(* IEC 61131-3 sources: astools/Data/ASTemplates/Default/Export Dialog/LogicalView/Libraries/FileIO, 3 files *)

(* ---- FileIO.typ ---- *)
TYPE
    fiDIR_READ_DATA		: STRUCT						(*directory read structure*)
        Filename		: ARRAY[0..259] OF USINT;		(*file name*)
        Date			: DATE_AND_TIME;				(*date and time*)
        Filelength		: UDINT;						(*file length*)
	END_STRUCT;

    fiDIR_READ_EX_DATA	: STRUCT						(*directory read extended structure*)
        Filename		: ARRAY[0..259] OF USINT;		(*file name*)
        Date			: DATE_AND_TIME;				(*date and time*)
        Filelength		: UDINT;						(*file length*)
        Mode			: UINT;							(*mode*)
	END_STRUCT;

	fiFILE_INFO			: STRUCT						(*file information structure*)
		size			: UDINT;						(*size of file [bytes]*)
		linkCnt			: UDINT;						(*link count*)
		accTime			: DATE_AND_TIME;				(*time of last access*)
		modTime			: DATE_AND_TIME;				(*time of last data modification*)
		chgTime			: DATE_AND_TIME;				(*time of last file status change*)
		reserved		: ARRAY[0..20] OF UDINT;		(*reserved for future use*)
	END_STRUCT;
END_TYPE

(* ---- FileIO.fun ---- *)
{REDUND_CONTEXT} {REDUND_UNREPLICABLE} FUNCTION_BLOCK FileCreate				(*creates a file; asynchronous execution*)
	VAR_INPUT
		enable		: BOOL;				(*enables execution*)
		pDevice		: UDINT;			(*device name given as a pointer*)
		pFile		: UDINT;			(*pointer to the file name*)
	END_VAR

	VAR
        i_state		: UINT;				(*internal variable*)
		i_result	: UINT;				(*internal variable*)
        i_tmp		: UDINT;			(*internal variable*)
	END_VAR

	VAR_OUTPUT
		status		: UINT;				(*execution status: ERR_OK, ERR_FUB_ENABLE_FALSE, ERR_FUB_BUSY, 0xXXXX = see help*)
		ident		: UDINT;			(*identifier of the created file*)
	END_VAR
END_FUNCTION_BLOCK

{REDUND_CONTEXT} {REDUND_UNREPLICABLE} FUNCTION_BLOCK FileOpen					(*opens a file; asynchronous execution*)
	VAR_INPUT
		enable		: BOOL;				(*enables execution*)
		pDevice		: UDINT;			(*device name given as a pointer*)
		pFile		: UDINT;			(*pointer to the file name*)
		mode		: USINT;			(*access mode (FILE_R, FILE_W, FILE_RW)*)
	END_VAR

	VAR
        i_state		: UINT;				(*internal variable*)
		i_result	: UINT;				(*internal variable*)
        i_tmp		: UDINT;			(*internal variable*)
	END_VAR

	VAR_OUTPUT
		status		: UINT;				(*execution status: ERR_OK, ERR_FUB_ENABLE_FALSE, ERR_FUB_BUSY, 0xXXXX = see help*)
		ident		: UDINT;			(*identifier of the created file*)
		filelen		: UDINT;			(*file length*)
	END_VAR
END_FUNCTION_BLOCK

{REDUND_CONTEXT} {REDUND_UNREPLICABLE} FUNCTION_BLOCK FileClose				(*closes an open file; asynchronous execution*)
	VAR_INPUT
		enable		: BOOL;				(*enables execution*)
		ident		: UDINT;			(*identifier of the created file*)
	END_VAR

	VAR
        i_state		: UINT;				(*internal variable*)
		i_result	: UINT;				(*internal variable*)
        i_tmp		: UDINT;			(*internal variable*)
	END_VAR

	VAR_OUTPUT
		status		: UINT;				(*execution status: ERR_OK, ERR_FUB_ENABLE_FALSE, ERR_FUB_BUSY, 0xXXXX = see help*)
	END_VAR
END_FUNCTION_BLOCK

{REDUND_CONTEXT} {REDUND_UNREPLICABLE} FUNCTION_BLOCK FileRead					(*reads from an open file; asynchronous execution*)
	VAR_INPUT
		enable		: BOOL;				(*enables execution*)
		ident		: UDINT;			(*identifier of the created file*)
		offset		: UDINT;			(*offset*)
		pDest		: UDINT;			(*pointer to the read buffer*)
		len			: UDINT;			(*length of bytes to read*)
	END_VAR

	VAR
        i_state		: UINT;				(*internal variable*)
		i_result	: UINT;				(*internal variable*)
        i_tmp		: UDINT;			(*internal variable*)
	END_VAR

	VAR_OUTPUT
		status		: UINT;				(*execution status: ERR_OK, ERR_FUB_ENABLE_FALSE, ERR_FUB_BUSY, 0xXXXX = see help*)
	END_VAR
END_FUNCTION_BLOCK

{REDUND_CONTEXT} {REDUND_UNREPLICABLE} FUNCTION_BLOCK FileReadEx				(*reads from an open file and returns the number of actually read bytes; asynchronous execution*)
	VAR_INPUT
		enable		: BOOL;				(*enables execution*)
		ident		: UDINT;			(*identifier of the created file*)
		offset		: UDINT;			(*offset*)
		pDest		: UDINT;			(*pointer to the read buffer*)
		len			: UDINT;			(*number of bytes to read*)
	END_VAR

	VAR
        i_state		: UINT;				(*internal variable*)
		i_result	: UINT;				(*internal variable*)
        i_tmp		: UDINT;			(*internal variable*)
	END_VAR

	VAR_OUTPUT
		status		: UINT;				(*execution status: ERR_OK, ERR_FUB_ENABLE_FALSE, ERR_FUB_BUSY, 0xXXXX = see help*)
		bytesread	: UDINT;			(*number of bytes read*)
	END_VAR
END_FUNCTION_BLOCK

{REDUND_CONTEXT} {REDUND_UNREPLICABLE} FUNCTION_BLOCK FileWrite				(*writes to a file; asynchronous execution*)
	VAR_INPUT
		enable		: BOOL;				(*enables execution*)
		ident		: UDINT;			(*identifier of the created file*)
		offset		: UDINT;			(*offset*)
		pSrc		: UDINT;			(*pointer to the write buffer*)
		len			: UDINT;			(*number of bytes to write*)
	END_VAR

	VAR
        i_state		: UINT;				(*internal variable*)
		i_result	: UINT;				(*internal variable*)
        i_tmp		: UDINT;			(*internal variable*)
	END_VAR

	VAR_OUTPUT
		status		: UINT;				(*execution status: ERR_OK, ERR_FUB_ENABLE_FALSE, ERR_FUB_BUSY, 0xXXXX = see help*)
	END_VAR
END_FUNCTION_BLOCK

{REDUND_CONTEXT} {REDUND_UNREPLICABLE} FUNCTION_BLOCK FileWriteEx				(*writes to a file; asynchronous execution*)
	VAR_INPUT
		enable		: BOOL;				(*enables execution*)
		ident		: UDINT;			(*identifier of the created file*)
		offset		: UDINT;			(*offset*)
		pSrc		: UDINT;			(*pointer to the write buffer*)
		len			: UDINT;			(*number of bytes to write*)
		option		: UDINT;			(*options*)
	END_VAR

	VAR
        i_state		: UINT;				(*internal variable*)
		i_result	: UINT;				(*internal variable*)
        i_tmp		: UDINT;			(*internal variable*)
	END_VAR

	VAR_OUTPUT
		status		: UINT;				(*execution status: ERR_OK, ERR_FUB_ENABLE_FALSE, ERR_FUB_BUSY, 0xXXXX = see help*)
	END_VAR
END_FUNCTION_BLOCK

{REDUND_CONTEXT} {REDUND_UNREPLICABLE} FUNCTION_BLOCK FileRename				(*renames files; asynchronous execution*)
	VAR_INPUT
		enable		: BOOL;				(*enables execution*)
		pDevice		: UDINT;			(*device name given as a pointer*)
		pName		: UDINT;			(*pointer to the file name*)
		pNewName	: UDINT;			(*pointer to the new file name*)
	END_VAR

	VAR
        i_state		: UINT;				(*internal variable*)
		i_result	: UINT;				(*internal variable*)
        i_tmp		: UDINT;			(*internal variable*)
	END_VAR

	VAR_OUTPUT
		status		: UINT;				(*execution status: ERR_OK, ERR_FUB_ENABLE_FALSE, ERR_FUB_BUSY, 0xXXXX = see help*)
	END_VAR
END_FUNCTION_BLOCK

{REDUND_CONTEXT} {REDUND_UNREPLICABLE} FUNCTION_BLOCK FileCopy					(*copies a file; asynchronous execution*)
	VAR_INPUT
		enable		: BOOL;				(*enables execution*)
		pSrcDev		: UDINT;			(*pointer to the source file device name*)
		pSrc		: UDINT;			(*pointer to the existing file name*)
		pDestDev	: UDINT;			(*pointer to the destination file device name*)
		pDest		: UDINT;			(*pointer to the copy file name*)
		option		: USINT;			(*copy option*)
	END_VAR

	VAR
        i_state		: UINT;				(*internal variable*)
		i_result	: UINT;				(*internal variable*)
        i_tmp		: UDINT;			(*internal variable*)
	END_VAR

	VAR_OUTPUT
		status		: UINT;				(*execution status: ERR_OK, ERR_FUB_ENABLE_FALSE, ERR_FUB_BUSY, 0xXXXX = see help*)
	END_VAR
END_FUNCTION_BLOCK

{REDUND_CONTEXT} {REDUND_UNREPLICABLE} FUNCTION_BLOCK FileDelete				(*deletes a file; asynchronous execution*)
	VAR_INPUT
		enable		: BOOL;				(*enables execution*)
		pDevice		: UDINT;			(*device name given as a pointer*)
		pName		: UDINT;			(*pointer to the file name*)
	END_VAR

	VAR
        i_state		: UINT;				(*internal variable*)
		i_result	: UINT;				(*internal variable*)
        i_tmp		: UDINT;			(*internal variable*)
	END_VAR

	VAR_OUTPUT
		status		: UINT;				(*execution status: ERR_OK, ERR_FUB_ENABLE_FALSE, ERR_FUB_BUSY, 0xXXXX = see help*)
	END_VAR
END_FUNCTION_BLOCK

{REDUND_CONTEXT} {REDUND_UNREPLICABLE} FUNCTION_BLOCK FileInfo					(*gets information about a file; asynchronous execution*)
	VAR_INPUT
		enable		: BOOL;				(*enables execution*)
		pDevice		: UDINT;			(*device name given as a pointer*)
		pName		: UDINT;			(*file name given as pointer*)
		pInfo		: UDINT;			(*file information (fiFILE_INFO) structure given as pointer*)
	END_VAR

	VAR
        i_state		: UINT;				(*internal variable*)
		i_result	: UINT;				(*internal variable*)
        i_tmp		: UDINT;			(*internal variable*)
	END_VAR

	VAR_OUTPUT
		status		: UINT;				(*execution status: ERR_OK, ERR_FUB_ENABLE_FALSE, ERR_FUB_BUSY, 0xXXXX = see help*)
	END_VAR
END_FUNCTION_BLOCK

{REDUND_CONTEXT} {REDUND_UNREPLICABLE} FUNCTION_BLOCK FileTruncate				(*truncates a file's length; asynchronous execution*)
	VAR_INPUT
		enable		: BOOL;				(*enables execution*)
		pDevice		: UDINT;			(*device name given as a pointer*)
		pName		: UDINT;			(*file name given as pointer*)
		newLength	: UDINT;			(*new length*)
	END_VAR

	VAR
        i_state		: UINT;				(*internal variable*)
		i_result	: UINT;				(*internal variable*)
        i_tmp		: UDINT;			(*internal variable*)
	END_VAR

	VAR_OUTPUT
		status		: UINT;				(*execution status: ERR_OK, ERR_FUB_ENABLE_FALSE, ERR_FUB_BUSY, 0xXXXX = see help*)
	END_VAR
END_FUNCTION_BLOCK

{REDUND_CONTEXT} {REDUND_UNREPLICABLE} FUNCTION_BLOCK DirCreate				(*creates a directory; asynchronous execution*)
	VAR_INPUT
		enable		: BOOL;				(*enables execution*)
		pDevice		: UDINT;			(*device name given as a pointer*)
		pName		: UDINT;			(*pointer to the directory name*)
	END_VAR

	VAR
        i_state		: UINT;				(*internal variable*)
		i_result	: UINT;				(*internal variable*)
        i_tmp		: UDINT;			(*internal variable*)
	END_VAR

	VAR_OUTPUT
		status		: UINT;				(*execution status: ERR_OK, ERR_FUB_ENABLE_FALSE, ERR_FUB_BUSY, 0xXXXX = see help*)
	END_VAR
END_FUNCTION_BLOCK

{REDUND_CONTEXT} {REDUND_UNREPLICABLE} FUNCTION_BLOCK DirOpen					(*opens a directory; asynchronous execution*)
	VAR_INPUT
		enable		: BOOL;				(*enables execution*)
		pDevice		: UDINT;			(*device name given as a pointer*)
		pName		: UDINT;			(*pointer to the directory name*)
	END_VAR

	VAR
        i_state		: UINT;				(*internal variable*)
		i_result	: UINT;				(*internal variable*)
        i_tmp		: UDINT;			(*internal variable*)
	END_VAR

	VAR_OUTPUT
		status		: UINT;				(*execution status: ERR_OK, ERR_FUB_ENABLE_FALSE, ERR_FUB_BUSY, 0xXXXX = see help*)
		ident		: UDINT;			(*identifier of the directory*)
	END_VAR
END_FUNCTION_BLOCK

{REDUND_CONTEXT} {REDUND_UNREPLICABLE} FUNCTION_BLOCK DirClose					(*closes a directory; asynchronous execution*)
	VAR_INPUT
		enable		: BOOL;				(*enables execution*)
		ident		: UDINT;			(*identifier of the directory*)
	END_VAR

	VAR
        i_state		: UINT;				(*internal variable*)
		i_result	: UINT;				(*internal variable*)
        i_tmp		: UDINT;			(*internal variable*)
	END_VAR

	VAR_OUTPUT
		status		: UINT;				(*execution status: ERR_OK, ERR_FUB_ENABLE_FALSE, ERR_FUB_BUSY, 0xXXXX = see help*)
	END_VAR
END_FUNCTION_BLOCK

{REDUND_CONTEXT} {REDUND_UNREPLICABLE} FUNCTION_BLOCK DirRead					(*reads the individual file names in a directory; asynchronous execution*)
	VAR_INPUT
		enable		: BOOL;				(*enables execution*)
		pDevice		: UDINT;			(*device name given as a pointer*)
		pPath		: UDINT;			(*pointer to the path string*)
		entry		: UDINT;			(*specifies which entry should be read*)
		option		: USINT;			(*specifies whether directory names or filenames should be read*)
		pData		: UDINT;			(*pointer to the memory area where the information is copied*)
		data_len	: UDINT;			(*length of the provided data area*)
	END_VAR

	VAR
        i_state		: UINT;				(*internal variable*)
		i_result	: UINT;				(*internal variable*)
        i_tmp		: UDINT;			(*internal variable*)
	END_VAR

	VAR_OUTPUT
		status		: UINT;				(*execution status: ERR_OK, ERR_FUB_ENABLE_FALSE, ERR_FUB_BUSY, 0xXXXX = see help*)
	END_VAR
END_FUNCTION_BLOCK

{REDUND_CONTEXT} {REDUND_UNREPLICABLE} FUNCTION_BLOCK DirReadEx				(*reads the individual file or directory names in a directory; asynchronous execution*)
	VAR_INPUT
		enable		: BOOL;				(*enables execution*)
		ident		: UDINT;			(*identifier of the directory*)
		pData		: UDINT;			(*pointer to the memory area where the information is copied*)
		data_len	: UDINT;			(*length of the available data area*)
	END_VAR

	VAR
        i_state		: UINT;				(*internal variable*)
		i_result	: UINT;				(*internal variable*)
        i_tmp		: UDINT;			(*internal variable*)
	END_VAR

	VAR_OUTPUT
		status		: UINT;				(*execution status: ERR_OK, ERR_FUB_ENABLE_FALSE, ERR_FUB_BUSY, 0xXXXX = see help*)
	END_VAR
END_FUNCTION_BLOCK

{REDUND_CONTEXT} {REDUND_UNREPLICABLE} FUNCTION_BLOCK DirInfo					(*gets information about a directory; asynchronous execution*)
	VAR_INPUT
		enable		: BOOL;				(*enables execution*)
		pDevice		: UDINT;			(*device name given as a pointer*)
		pPath		: UDINT;			(*pointer to the path (directory name)*)
	END_VAR

	VAR
        i_state		: UINT;				(*internal variable*)
		i_result	: UINT;				(*internal variable*)
        i_tmp		: UDINT;			(*internal variable*)
	END_VAR

	VAR_OUTPUT
		status		: UINT;				(*execution status: ERR_OK, ERR_FUB_ENABLE_FALSE, ERR_FUB_BUSY, 0xXXXX = see help*)
		dirnum		: UDINT;			(*number of subdirectories in this directory*)
		filenum		: UDINT;			(*number of files in this directory*)
	END_VAR
END_FUNCTION_BLOCK

{REDUND_CONTEXT} {REDUND_UNREPLICABLE} FUNCTION_BLOCK DirRename				(*renames directories; asynchronous execution*)
	VAR_INPUT
		enable		: BOOL;				(*enables execution*)
		pDevice		: UDINT;			(*device name given as a pointer*)
		pName		: UDINT;			(*pointer to the directory name*)
		pNewName	: UDINT;			(*pointer to the new directory name*)
	END_VAR

	VAR
        i_state		: UINT;				(*internal variable*)
		i_result	: UINT;				(*internal variable*)
        i_tmp		: UDINT;			(*internal variable*)
	END_VAR

	VAR_OUTPUT
		status		: UINT;				(*execution status: ERR_OK, ERR_FUB_ENABLE_FALSE, ERR_FUB_BUSY, 0xXXXX = see help*)
	END_VAR
END_FUNCTION_BLOCK

{REDUND_CONTEXT} {REDUND_UNREPLICABLE} FUNCTION_BLOCK DirCopy					(*copies a directory*)
	VAR_INPUT
		enable		: BOOL;				(*enables execution*)
		pSrcDev		: UDINT;			(*pointer to the source file device name*)
		pSrcDir		: UDINT;			(*pointer to the source directory name*)
		pDestDev	: UDINT;			(*pointer to the destination file device name*)
		pDestDir	: UDINT;			(*pointer to the destination directory name*)
		option		: USINT;			(*copy option*)
	END_VAR

	VAR
        i_state		: UINT;				(*internal variable*)
		i_result	: UINT;				(*internal variable*)
        i_tmp		: UDINT;			(*internal variable*)
	END_VAR

	VAR_OUTPUT
		status		: UINT;				(*execution status: ERR_OK, ERR_FUB_ENABLE_FALSE, 0xXXXX = see help*)
	END_VAR
END_FUNCTION_BLOCK

{REDUND_CONTEXT} {REDUND_UNREPLICABLE} FUNCTION_BLOCK DirDelete				(*deletes a directory; asynchronous execution*)
	VAR_INPUT
		enable		: BOOL;				(*enables execution*)
		pDevice		: UDINT;			(*device name given as a pointer*)
		pName		: UDINT;			(*pointer to the directory name*)
	END_VAR

	VAR
        i_state		: UINT;				(*internal variable*)
		i_result	: UINT;				(*internal variable*)
        i_tmp		: UDINT;			(*internal variable*)
	END_VAR

	VAR_OUTPUT
		status		: UINT;				(*execution status: ERR_OK, ERR_FUB_ENABLE_FALSE, ERR_FUB_BUSY, 0xXXXX = see help*)
	END_VAR
END_FUNCTION_BLOCK

{REDUND_CONTEXT} {REDUND_UNREPLICABLE} FUNCTION_BLOCK DirDeleteEx				(*deletes a directory (all files and subdirectories); asynchronous execution*)
	VAR_INPUT
		enable		: BOOL;				(*enables execution*)
		pDevice		: UDINT;			(*device name given as a pointer*)
		pName		: UDINT;			(*pointer to the directory name*)
	END_VAR

	VAR
        i_state		: UINT;				(*internal variable*)
		i_result	: UINT;				(*internal variable*)
        i_tmp		: UDINT;			(*internal variable*)
	END_VAR

	VAR_OUTPUT
		status		: UINT;				(*execution status: ERR_OK, ERR_FUB_ENABLE_FALSE, ERR_FUB_BUSY, 0xXXXX = see help*)
	END_VAR
END_FUNCTION_BLOCK

{REDUND_CONTEXT} {REDUND_UNREPLICABLE} FUNCTION_BLOCK SetAttributes			(*sets attributes; asynchronous execution*)
	VAR_INPUT
		enable		: BOOL;				(*enables execution*)
		pDevice		: UDINT;			(*device name given as a pointer*)
		pPath		: UDINT;			(*pointer to the path name (file or directory)*)
		attributes	: USINT;			(*attributes*)
		option		: USINT;			(*set options*)
	END_VAR

	VAR
        i_state		: UINT;				(*internal variable*)
		i_result	: UINT;				(*internal variable*)
        i_tmp		: UDINT;			(*internal variable*)
	END_VAR

	VAR_OUTPUT
		status		: UINT;				(*execution status: ERR_OK, ERR_FUB_ENABLE_FALSE, ERR_FUB_BUSY, 0xXXXX = see help*)
	END_VAR
END_FUNCTION_BLOCK

{REDUND_CONTEXT} {REDUND_UNREPLICABLE} FUNCTION_BLOCK GetAttributes			(*reads attributes; asynchronous execution*)
	VAR_INPUT
		enable		: BOOL;				(*enables execution*)
		pDevice		: UDINT;			(*device name given as a pointer*)
		pPath		: UDINT;			(*pointer to the path name (file or directory)*)
	END_VAR

	VAR
        i_state		: UINT;				(*internal variable*)
		i_result	: UINT;				(*internal variable*)
        i_tmp		: UDINT;			(*internal variable*)
	END_VAR

	VAR_OUTPUT
		status		: UINT;				(*execution status: ERR_OK, ERR_FUB_ENABLE_FALSE, ERR_FUB_BUSY, 0xXXXX = see help*)
		attributes	: USINT;			(*attributes*)
	END_VAR
END_FUNCTION_BLOCK

{REDUND_CONTEXT} {REDUND_UNREPLICABLE} FUNCTION_BLOCK DevMemInfo				(*determines a file device's memory information; asynchronous execution*)
	VAR_INPUT
		enable		: BOOL;				(*enables execution*)
		pDevice		: UDINT;			(*device name given as a pointer*)
	END_VAR

	VAR
        i_state		: UINT;				(*internal variable*)
		i_result	: UINT;				(*internal variable*)
        i_tmp		: UDINT;			(*internal variable*)
	END_VAR

	VAR_OUTPUT
		status		: UINT;				(*execution status: ERR_OK, ERR_FUB_ENABLE_FALSE, ERR_FUB_BUSY, 0xXXXX = see help*)
		freemem		: UDINT;			(*available disk space*)
		memsize		: UDINT;			(*total disk space*)
	END_VAR
END_FUNCTION_BLOCK

{REDUND_CONTEXT} {REDUND_UNREPLICABLE} FUNCTION_BLOCK DevLink					(*creates the file device; asynchronous execution*)
	VAR_INPUT
		enable		: BOOL;				(*enables execution*)
		pDevice		: UDINT;			(*new device name given as a pointer*)
		pParam		: UDINT;			(*pointer to the link parameter*)
	END_VAR

	VAR
        i_state		: UINT;				(*internal variable*)
		i_result	: UINT;				(*internal variable*)
        i_tmp		: UDINT;			(*internal variable*)
	END_VAR

	VAR_OUTPUT
		status		: UINT;				(*execution status: ERR_OK, ERR_FUB_ENABLE_FALSE, ERR_FUB_BUSY, 0xXXXX = see help*)
		handle		: UDINT;			(*file device handle*)
	END_VAR
END_FUNCTION_BLOCK

{REDUND_CONTEXT} {REDUND_UNREPLICABLE} FUNCTION_BLOCK DevUnlink				(*unlinks the device; asynchronous execution*)
	VAR_INPUT
		enable		: BOOL;				(*enables execution*)
		handle		: UDINT;			(*file device handle*)
	END_VAR

	VAR
        i_state		: UINT;				(*internal variable*)
		i_result	: UINT;				(*internal variable*)
        i_tmp		: UDINT;			(*internal variable*)
	END_VAR

	VAR_OUTPUT
		status		: UINT;				(*execution status: ERR_OK, ERR_FUB_ENABLE_FALSE, ERR_FUB_BUSY, 0xXXXX = see help*)
	END_VAR
END_FUNCTION_BLOCK

{REDUND_CONTEXT} {REDUND_UNREPLICABLE} FUNCTION_BLOCK GetVolumeLabel			(*reads volume label; asynchronous execution*)
	VAR_INPUT
		enable		: BOOL;				(*enables execution*)
		pDevice		: UDINT;			(*device name given as a pointer*)
		pLabel		: UDINT;			(*buffer for volume label given as pointer*)
		labelMax	: UDINT;			(*size of buffer for volume label*)
	END_VAR

	VAR
        i_state		: UINT;				(*internal variable*)
		i_result	: UINT;				(*internal variable*)
        i_tmp		: UDINT;			(*internal variable*)
	END_VAR

	VAR_OUTPUT
		status		: UINT;				(*execution status: ERR_OK, ERR_FUB_ENABLE_FALSE, ERR_FUB_BUSY, 0xXXXX = see help*)
		labelLen	: UDINT;			(*length of volume label*)
	END_VAR
END_FUNCTION_BLOCK

{REDUND_CONTEXT} {REDUND_UNREPLICABLE} FUNCTION_BLOCK GetVolumeSerialNo		(*reads volume serial nummer; asynchronous execution*)
	VAR_INPUT
		enable		: BOOL;				(*enables execution*)
		pDevice		: UDINT;			(*device name given as a pointer*)
	END_VAR

	VAR
        i_state		: UINT;				(*internal variable*)
		i_result	: UINT;				(*internal variable*)
        i_tmp		: UDINT;			(*internal variable*)
	END_VAR

	VAR_OUTPUT
		status		: UINT;				(*execution status: ERR_OK, ERR_FUB_ENABLE_FALSE, ERR_FUB_BUSY, 0xXXXX = see help*)
		serialNo	: UDINT;			(*volume serialNo*)
	END_VAR
END_FUNCTION_BLOCK

FUNCTION FileIoGetSysError	: UINT		(*reads system errors*)
END_FUNCTION

(* ---- FileIO.var ---- *)
VAR CONSTANT
	fiATTR_ARCHIVE					: USINT := 32;			(*attribute archive*)
	fiATTR_DIRECTORY				: USINT := 16;			(*attribute directory*)
	fiATTR_HIDDEN 					: USINT := 2;			(*attribute hidden*)
	fiATTR_RDONLY 					: USINT := 1;			(*attribute read only*)
	fiATTR_SYSTEM 					: USINT := 4;			(*attribute system*)
	fiATTR_VOL_LABEL 				: USINT := 8;			(*attribute volume label*)

	fiRECURSIVE						: USINT := 1;			(*option recursive*)
	fiOVERWRITE						: USINT := 2;			(*option overwrite*)

	fiREAD_ONLY 					: USINT := 0;			(*access mode read only*)
	fiWRITE_ONLY 					: USINT := 1;			(*access mode write only*)
	fiREAD_WRITE 					: USINT := 2;			(*access mode read and write*)

	fiFILE							: USINT := 0;			(*directory read files only*)
	fiDIRECTORY						: USINT := 1;			(*directory read directories only*)
	fiBOTH							: USINT := 2;			(*directory read files and directories*)

	fiTruncate						: UDINT := 1;			(*truncate file*)

	fiERR_INVALID_PATH  			: UINT := 20700;		(*error invalid path*)
	fiERR_DATA_SIZE  				: UINT := 20701;		(*error data size*)
	fiERR_NO_MORE_ENTRIES  			: UINT := 20702;		(*error no more entries*)
	fiERR_NOT_SUPPORTED  			: UINT := 20703;		(*error not supported*)
	fiERR_INVALID_TYP 				: UINT := 20704;		(*error invalid type*)
	fiERR_EXIST  					: UINT := 20705;		(*error exist*)
	fiERR_ACCESS 					: UINT := 20706;		(*error access*)
	fiERR_MODE  					: UINT := 20707;		(*error mode*)
	fiERR_FILE_NOT_FOUND  			: UINT := 20708;		(*error file not found*)
	fiERR_FILE_DEVICE  				: UINT := 20709;		(*error file device*)
	fiERR_SPACE  					: UINT := 20710;		(*error space*)
	fiERR_SEEK  					: UINT := 20711;		(*error seek*)
	fiERR_FILE  					: UINT := 20712;		(*error file*)
	fiERR_LESS_VIRTUAL_MEMORY  		: UINT := 20713;		(*error less virtual memory*)
	fiERR_COM_FILE_OPEN  			: UINT := 20714;		(*error file open*)
	fiERR_COM_FILE_CLOSE  			: UINT := 20715;		(*error file close*)
	fiERR_COM_FILE_READ  			: UINT := 20716;		(*error file read*)
	fiERR_COM_FILE_WRITE  			: UINT := 20717;		(*error file write*)
	fiERR_COM_FILE_IOCTL  			: UINT := 20718;		(*error fiel ioctl*)
	fiERR_DATA  					: UINT := 20719;		(*error data*)
	fiERR_ASYNC_MANAGER  			: UINT := 20720;		(*error asynchron manager*)
	fiERR_FILE_NOT_OPENED  			: UINT := 20721;		(*error file not opened*)
	fiERR_INVALID_DIRECTORY  		: UINT := 20722;		(*error invalid directory*)
	fiERR_DIR_NOT_EXIST  			: UINT := 20723;		(*error directory not exists*)
	fiERR_DIR_NOT_EMPTY  			: UINT := 20724;		(*error directory not empty*)
	fiERR_DIR_ALREADY_EXIST 		: UINT := 20725;		(*error directory already exists*)
	fiERR_DETMEMINFO  				: UINT := 20726;		(*error dedect memory info*)
	fiERR_NOT_ENOUGH_FREEMEM  		: UINT := 20727;		(*error not enough free memory*)
	fiERR_DIR_INVALID_HANDLE		: UINT := 20728;		(*error invalid directory handle*)
	fiERR_PARAMETER  				: UINT := 20729;		(*error parameter*)
	fiERR_DEVICE_ALREADY_EXIST		: UINT := 20730;		(*error device already exists*)
	fiERR_DEVICE_INVALID_HANDLE		: UINT := 20731;		(*error invalid device handle*)
	fiERR_NETIO_IP_UNEQUAL			: UINT := 20732;		(*ungleiche IP bei identischem Hostnamen - IP-overwrite nicht gesetzt*)
	fiERR_NETIO_PORT				: UINT := 20733;		(*error port not supported*)
	fiERR_NETIO_USER				: UINT := 20734;		(*error user or password*)
	fiERR_INVALID_NBYTES			: UINT := 20735;		(*error invalid number of bytes*)
	fiERR_NETIO_PARAMETERS			: UINT := 20736;		(*error invalid parameters to establish a connection*)

	fiERR_INIT  					: UINT := 20796;		(*error init*)
	fiERR_DEVICE_DRIVER  			: UINT := 20797;		(*error device driver*)
	fiERR_DEVICE_MANAGER  			: UINT := 20798;		(*error device manager*)
	fiERR_SYSTEM  					: UINT := 20799;		(*error system*)

	ATTR_ARCHIVE					: USINT := 32;			(*obsolete*)
	ATTR_DIRECTORY					: USINT := 16;			(*obsolete*)
	ATTR_HIDDEN						: USINT := 2;			(*obsolete*)
	ATTR_RDONLY						: USINT := 1;			(*obsolete*)
	ATTR_SYSTEM						: USINT := 4;			(*obsolete*)
	ATTR_VOL_LABEL					: USINT := 8;			(*obsolete*)
	DIR_OW							: USINT := 1;			(*obsolete*)
	FILE_ALL						: USINT := 2;			(*obsolete*)
	FILE_DIR						: USINT := 1;			(*obsolete*)
	FILE_FILE						: USINT := 0;			(*obsolete*)
	FILE_ONCE						: USINT := 0;			(*obsolete*)
	FILE_DETMEM						: USINT := 1;			(*obsolete*)
	FILE_OW_DETMEM					: USINT := 2;			(*obsolete*)
	FILE_OW_ONCE					: USINT := 3;			(*obsolete*)
	FILE_R							: USINT := 0;			(*obsolete*)
	FILE_W							: USINT := 1;			(*obsolete*)
	FILE_RW							: USINT := 2;			(*obsolete*)
	SET_RECURSIVE					: USINT := 1;			(*obsolete*)
END_VAR
